{attribute 'qualified_only'}
{attribute 'strict'}
{attribute 'to_string'}
TYPE E_FsmError :
(
	NO_ERR		  := 0,
	INIT_ERR      := 1,
	STAT_ERR      := 2,
	STAT_TR_ERR   := 3,
	NOM_LEV_ERR   := 4,
	INTER_TR_ERR  := 5,
	END_TR_ERR    := 6
);
END_TYPE

(* stored: Version 1.1.0.1, ProductVersion 3.1.4024.12
   DUT E_FsmError: Id {eb4858ad-2204-4f10-8045-2a371bb87cbc} *)
